(*

.. <legal notes>

legal notes
=================
| SPDX-FileCopyrightText: © 2025 Oleksandr Tiutyk <trofimich@gmail.com>
| SPDX-License-Identifier: LGPL-3.0-only
| For details check: LGPL-3.0-only_

.. _LGPL-3.0-only: https://www.gnu.org/licenses/lgpl-3.0.en.html

.. </legal notes>

*)

INTERFACE IGenericConversionNotSupportedException EXTENDS IGeneralException

END_INTERFACE

(* stored: Version 1.1.0.1
   Itf IGenericConversionNotSupportedException: Id {67a2a108-d3bc-4b19-a1e1-b16c2025427d} *)
